// TIA Portal V18 export
TYPE "UDT_DOadv"
// stored: IsFailsafeCompliant false
   STRUCT
      xInput : Bool;   // Value for DO
      xOutput : Bool;   // Phisicl output
      xMemoryIn : Bool;   // Internal
      xInversion : Bool;
      xMemoryOut : Bool;
      xReserv3 : Bool;
      xReserv4 : Bool;
      xReserv5 : Bool;
      iCounterIn : Int;   // Counter
      iCounterOut : Int;
      iFuncSystemID : Byte := 0;
      iFuncVar : Byte := 0;
      cMOA : Byte;   // Mode Manual/Off/Auto
      cMemory : Byte;
   END_STRUCT;
END_TYPE
